// TIA Portal V20 export
// export: Created 2025-12-01T14:57:16.4921302Z, ExportSetting None, DisplayName Totally Integrated Automation Portal, DisplayVersion V20 Update 3, DisplayName TIA Portal Openness, DisplayVersion V20 Update 3, DisplayName TIA Portal Version Control Interface, DisplayVersion V20 Update 3, DisplayName STEP 7 Professional, DisplayVersion V20 Update 3, DisplayName STEP 7 Safety, DisplayVersion V20 Update 2, DisplayName WinCC Basic/Comfort/Advanced, DisplayVersion V20 Update 3, DisplayName WinCC Professional, DisplayVersion V20 Update 3, DisplayName WinCC Unified, DisplayVersion V20 Update 3
DATA_BLOCK "DB891_VariablesTCP"   // DB891
{ S7_Optimized_Access := 'FALSE' }
AUTHOR : TRACKING
NAME : 20130301
VERSION : 3.0
// stored: AutoNumber false
   VAR
      TCON_JdT_PLC_Req : Bool;
      TCON_JdT_PLC_Done : Bool;
      TCON_JdT_PLC_Busy : Bool;
      TCON_JdT_PLC_Error : Bool;
      TCON_JdT_PLC_Flanco : Bool;
      Bit_05 : Bool;
      Bit_06 : Bool;
      Bit_07 : Bool;
      TDISCON_JdT_PLC_Req : Bool;
      TDISCON_JdT_PLC_Done : Bool;
      TDISCON_JdT_PLC_Busy : Bool;
      TDISCON_JdT_PLC_Error : Bool;
      TDISCON_JdT_PLC_Flanco : Bool;
      Bit_15 : Bool;
      Bit_16 : Bool;
      Bit_17 : Bool;
      TSEND_JdT_PLC_Req : Bool := TRUE;
      TSEND_JdT_PLC_Done : Bool;
      TSEND_JdT_PLC_Busy : Bool;
      TSEND_JdT_PLC_Error : Bool;
      TSEND_JdT_PLC_Flanco : Bool;
      Bit_25 : Bool;
      Bit_26 : Bool;
      Bit_27 : Bool;
      TRCV_JdT_PLC_Req : Bool;
      TRCV_JdT_PLC_Done : Bool;
      TRCV_JdT_PLC_Busy : Bool;
      TRCV_JdT_PLC_Error : Bool;
      Bit_34 : Bool;
      Bit_35 : Bool;
      Bit_36 : Bool;
      Bit_37 : Bool;
      TCON_JdT_PLC_Status : Word;
      TDISCON_JdT_PLC_Status : Word;
      TSEND_JdT_PLC_Status : Word;
      TRCV_JdT_PLC_Status : Word;
      TCON_JdT_PLC_MStatus : Word;
      TDISCON_JdT_PLC_MStatus : Word;
      TSEND_JdT_PLC_MStatus : Word;
      TRCV_JdT_PLC_MStatus : Word;
      TSEND_JdT_PLC_Longitud : Int;
      TRCV_JdT_PLC_Longitud : Int;
      TCON_JdT_PLC_Req_JDT02 : Bool;
      TCON_JdT_PLC_Done_JDT02 : Bool;
      TCON_JdT_PLC_Busy_JDT02 : Bool;
      TCON_JdT_PLC_Error_JDT02 : Bool;
      TCON_JdT_PLC_Flanco_JDT02 : Bool;
      Bit_6 : Bool;
      Bit_7 : Bool;
      Bit_8 : Bool;
      TDISCON_JdT_PLC_Req_JDT02 : Bool;
      TDISCON_JdT_PLC_Done_JDT02 : Bool;
      TDISCON_JdT_PLC_Busy_JDT02 : Bool;
      TDISCON_JdT_PLC_Error_JDT02 : Bool;
      TDISCON_JdT_PLC_Flanco_JDT02 : Bool;
      Bit_18 : Bool;
      Bit_19 : Bool;
      Bit_20 : Bool;
      TSEND_JdT_PLC_Req_JDT02 : Bool := TRUE;
      TSEND_JdT_PLC_Done_JDT02 : Bool;
      TSEND_JdT_PLC_Busy_JDT02 : Bool;
      TSEND_JdT_PLC_Error_JDT02 : Bool;
      TSEND_JdT_PLC_Flanco_JDT02 : Bool;
      Bit_28 : Bool;
      Bit_29 : Bool;
      Bit_30 : Bool;
      TRCV_JdT_PLC_Req_JDT02 : Bool;
      TRCV_JdT_PLC_Done_JDT02 : Bool;
      TRCV_JdT_PLC_Busy_JDT02 : Bool;
      TRCV_JdT_PLC_Error_JDT02 : Bool;
      Bit_38 : Bool;
      Bit_39 : Bool;
      Bit_40 : Bool;
      Bit_41 : Bool;
      TCON_JdT_PLC_Status_JDT02 : Word;
      TDISCON_JdT_PLC_Status_JDT02 : Word;
      TSEND_JdT_PLC_Status_JDT02 : Word;
      TRCV_JdT_PLC_Status_JDT02 : Word;
      TCON_JdT_PLC_MStatus_JDT02 : Word;
      TDISCON_JdT_PLC_MStatus_JDT02 : Word;
      TSEND_JdT_PLC_MStatus_JDT02 : Word;
      TRCV_JdT_PLC_MStatus_JDT02 : Word;
      TSEND_JdT_PLC_Longitud_JDT02 : Int;
      TRCV_JdT_PLC_Longitud_JDT02 : Int;
   END_VAR
BEGIN
END_DATA_BLOCK
